Fanuc KAREL source: kt00184.KL

PROGRAM KT00184
%NOLOCKGROUP
VAR
Y1 : ARRAY[2] OF BYTE
H2 : ARRAY[2] OF SHORT
OUT:REAL
BEGIN
Y1[1]=2
H2[1]=3
OUT=((Y1[1] MOD H2[1]))
END KT00184
